// LS Electric XG5000 project: 2023-09-04 #1
// PLC NewPLC
// module base 0 slot 0: 입출력 모듈:XBC-DR32H (DC 24V 입력, 릴레이 출력 32점)

PROGRAM NewProgram (task: 스캔 프로그램)

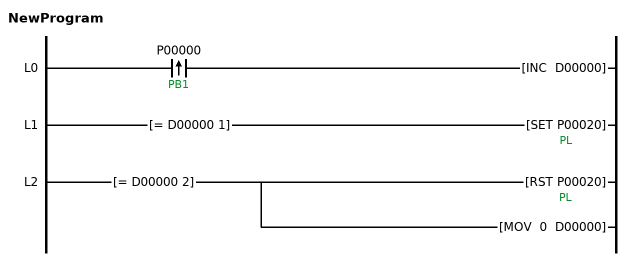
; L0
LOADP     P00000	// PB1
INC       D00000
; L1
LOAD=     D00000 1
SET       P00020	// PL
; L2
LOAD=     D00000 2
RST       P00020	// PL
MOV       0 D00000